// Hardware-linked primitives for FB_AnalogOutput. A 32-bit UNION covers
// every common EL4xxx terminal — 4-20 mA, 0-10 V, 16-bit DAC, 32-bit
// positioner, etc. Choose the numeric interpretation with cfg.cfgOutputType.
//
// Link at instance site via
//     {attribute 'TcLinkTo' := '.io.outRaw.dw := TIID^...^Output'}
//
// See docs/8-IO-Binding.md for the full worked examples.
TYPE ST_AnalogOutput_IO :
STRUCT
    outRaw : U_IoRaw_Out;
END_STRUCT
END_TYPE

(* stored: Version 1.1.0.1, ProductVersion 3.1.4026.12
   DUT ST_AnalogOutput_IO: Id {b0100004-0003-0000-0000-000000000001} *)
